// TIA Portal V17 export
// export: Created 2022-07-04T15:11:30.0499403Z, ExportSetting WithDefaults, DisplayName Totally Integrated Automation Portal, DisplayVersion V17, DisplayName TIA Portal Openness, DisplayVersion V17, DisplayName TIA Portal Version Control Interface, DisplayVersion V17, DisplayName STEP 7 Professional, DisplayVersion V17, DisplayName STEP 7 Safety, DisplayVersion V17, DisplayName WinCC Advanced, DisplayVersion V17
DATA_BLOCK "ControllingInterface"   // DB5
{ S7_Optimized_Access := 'TRUE' }
VERSION : 0.1
// stored: AutoNumber true, DBAccessibleFromOPCUA true, DBAccessibleFromWebserver true, IsOnlyStoredInLoadMemory false, IsRetainMemResEnabled false, IsWriteProtectedInAS false, MemoryReserve 100
   VAR
      new { S7_SetPoint := 'True'} : Bool;
      opcUaConnect : Bool;
      opcUaRead : Bool;
      opcUaWrite : Bool;
      opcUaMethodCall : Bool;
      opcUaMethodIndex : SInt;
      opcUaConnected { S7_SetPoint := 'True'} : Bool;
      opcUaDone : Bool;
      opcUaBusy : Bool;
      opcUaError : Bool;
      opcUaStatus : Word;
      opcUaDiagnostics : "typeFbDiagnostics";
   END_VAR
BEGIN
END_DATA_BLOCK
